% RSLogix 500 project I2P JOB 27 - SOLUTION_BAK001.RSS, saved by version 10.00.00.00 %
PROJECT "UNTITLED"    % processor: Bul.1763 MicroLogix 1100 Series B %

PROGRAM FILES
  LAD 2   8 rungs

DATA FILES
  O0 OUTPUT  4 elements
  I1 INPUT  6 elements
  S2 STATUS  66 elements
  B3 BINARY  1 elements
  T4 TIMER  1 elements
  C5 COUNTER  1 elements
  R6 CONTROL  1 elements
  N7 INTEGER  1 elements
  F8 FLOAT  1 elements

LADDER 2
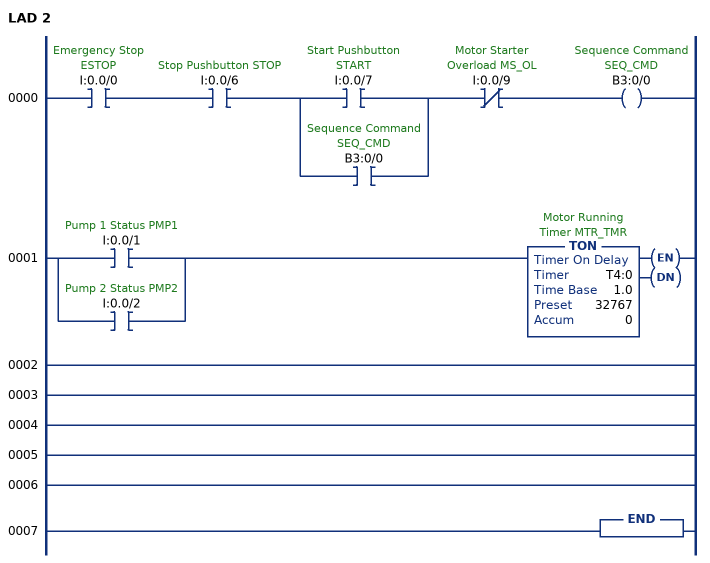
% Rung: 0 %  % edit flag set %
SOR XIC I:0.0/0 XIC I:0.0/6 BST XIC I:0.0/7 NXB XIC B3:0/0 BND XIO I:0.0/9 OTE B3:0/0 EOR
%   I:0.0/0  ESTOP  "Emergency Stop" %
%   I:0.0/6  STOP  "Stop Pushbutton" %
%   I:0.0/7  START  "Start Pushbutton" %
%   B3:0/0  SEQ_CMD  "Sequence Command" %
%   I:0.0/9  MS_OL  "Motor Starter Overload" %
% Rung: 1 %  % edit flag set %
SOR BST XIC I:0.0/1 NXB XIC I:0.0/2 BND TON T4:0 1.0 32767 0 EOR
%   I:0.0/1  PMP1  "Pump 1 Status" %
%   I:0.0/2  PMP2  "Pump 2 Status" %
%   T4:0  MTR_TMR  "Motor Running Timer" %
% Rung: 2 %  % edit flag set %
SOR EOR
% Rung: 3 %  % edit flag set %
SOR EOR
% Rung: 4 %  % edit flag set %
SOR EOR
% Rung: 5 %  % edit flag set %
SOR EOR
% Rung: 6 %  % edit flag set %
SOR EOR
% Rung: 7 %
SOR END EOR
